(* IEC 61131-3 sources: Lasal/CPU_5344_V01/Class/FubOnDelayTimer, 1 file *)

(* ---- FubOnDelayTimer.st ---- *)
(*!
<Class
	Name               = "FubOnDelayTimer"
	Revision           = "1.0"
	RealtimeTask       = "false"
	CyclicTask         = "false"
	BackgroundTask     = "false"
	Sigmatek           = "true"
	OSInterface        = "false"
	HighPriority       = "false"
	Automatic          = "false"
	UpdateMode         = "Prescan"
	SharedCommandTable = "true"
	Objectsize         = "(284,120)"
	Comment            = "The on-delay timer can be used to&#13;&#10;delay setting an output true, for&#13;&#10;a fixed period after an input becomes&#13;&#10;true.&#13;&#10; ">
	<Channels>
		<Server Name="sET" Visualized="false" Initialize="false" WriteProtected="true" Retentive="false" Comment="elapsed time in ms"/>
		<Server Name="sQ1" Visualized="false" Initialize="false" WriteProtected="true" Retentive="false" Comment="Output"/>
		<Client Name="cIN" Required="false" Internal="false" Comment="Input"/>
		<Client Name="cPT" Required="false" Internal="false" Comment="delaytime in ms"/>
	</Channels>
</Class>
*)
FubOnDelayTimer : CLASS
  //Servers:
	sQ1 	: SvrChCmd_DINT;
	sET 	: SvrCh_DINT;
  //Clients:
	cIN 	: CltCh_DINT;
	cPT 	: CltCh_DINT;
  //Variables:
		merker 	: BOOL;
		timemark 	: UDINT;
  //Functions:

	FUNCTION VIRTUAL GLOBAL sQ1::Read
		VAR_OUTPUT
			output (EAX) 	: DINT;
		END_VAR;
  //Tables:
	FUNCTION @STD
		VAR_OUTPUT
			ret_code	: CONFSTATES;
		END_VAR;
	FUNCTION GLOBAL TAB @CT_;
END_CLASS;

//[#ENGLISH]
// ******************************************************************
//          TON - On delay timer
// ******************************************************************
//			CLIENT:
//			    cIN: input
//					cPT: output time in ms
//      SERVER:
//          sQ:  output
//          sET: elapsed time in ms
//
//   description:
//   The on-delay timer can be used to delay setting an output true,
//   for a fixed period after an input becomes true.
//   As input cIN goes true, the elapsed time at output sET starts to
//   increase. When the elapsed time reaches the time specified by
//   the  input cPT, the output goes true, and the elapsed time is
//   held.
//   The output sQ remains true until the input cIN goes false. If
//   the input is not true longer than the delay time specified in
//   cPT, the output remains false.
//
// ******************************************************************
// 		 created 		:		 AG		 :   	KW 38/05
// ******************************************************************
//                operation of READ function
// ******************************************************************
//   tested: AW | 05.10.2005 | Lasal2 v02.01.020 |
// ******************************************************************

FUNCTION VIRTUAL GLOBAL FubOnDelayTimer::sQ1::Read
	VAR_OUTPUT
		output (EAX) 	: DINT;
	END_VAR

  cIN := cIN.read();

  if (cIN = 0) then // = RESET
    merker 		:= false;
    sQ1	:= 0;
    sET	:= 0;
	else
		if (merker = false) then
			merker 	 := true;           // set START and TRG+
			timemark := ops.tAbsolute;  // store Time
			cPT 	   := cPT.read();	    // reading channel
			if (cPT = 0) then
				sQ1 := cIN; // OUT set to IN
			end_if;
		else // Time is running
			sET := (ops.tAbsolute - timemark)$DINT;
			if (sET >= cPT | sQ1 <> 0) then
        sQ1 := cIN; // OUT set to IN
				sET := cPT;
				timemark := ops.tAbsolute - sET$UDINT;
			end_if;
		end_if;
	end_if;

	output := sQ1;

END_FUNCTION
